{attribute 'qualified_only'}
{attribute 'strict'}
TYPE E_RobotTCPReceive :
(
	Idle,
	Connect_Start,
	Connect_Wait,
	Receive_Start,
	Receive_Wait,
	ParseData,
	RecordData,
	RecordData_Wait,
	Close_Start,
	Close_Wait,
	HandleError
);
END_TYPE

(* stored: Version 1.1.0.1, ProductVersion 3.1.4020.12
   DUT E_RobotTCPReceive: Id {551317f7-4e08-402d-b29c-244a13308ac0} *)
